Fanuc TP program (LS listing): pick_and_place.ls

/PROG  PICK_AND_PLACE
/ATTR
OWNER		= MNEDITOR;
COMMENT		= "";
PROG_SIZE	= 5834;
CREATE		= DATE 26-07-14  TIME 16:19:38;
MODIFIED	= DATE 26-07-14  TIME 16:19:38;
FILE_NAME	= PICK_AND;
VERSION		= 0;
LINE_COUNT	= 270;
MEMORY_SIZE	= 6422;
PROTECT		= READ_WRITE;
TCD:  STACK_SIZE	= 0,
      TASK_PRIORITY	= 50,
      TIME_SLICE	= 0,
      BUSY_LAMP_OFF	= 0,
      ABORT_REQUEST	= 0,
      PAUSE_REQUEST	= 0;
DEFAULT_GROUP	= 1,*,*,*,*;
CONTROL_CODE	= 00000000 00000000;
LOCAL_REGISTERS	= 0,0,0;
/APPL
/APPL
/MN
   1:  ! Main driving loop ;
   2:  LBL[4:PP_LOOP] ;
   3:   ;
   4:  ! Reset Error Checking ;
   5:  R[24:PICK_CNT_ERR]=0    ;
   6:  R[25:PLACE_CNT_ERR]=0    ;
   7:   ;
   8:  ! Check for recipe reset ;
   9:  IF R[11:RECIPE_IO_IDX]=37,JMP LBL[998] ;
  10:  R[12:RECIPE_OUTPUT]=R[R[99]]    ;
  11:   ;
  12:  ! Checks next recipe output ;
  13:  IF R[12:RECIPE_OUTPUT]=0,JMP LBL[1] ;
  14:   ;
  15:  LBL[24] ;
  16:  ! get out of shroud safely ;
  17:J PR[20] 100% CNT30    ;
  18:   ;
  19:  ! Move to next pin ;
  20:J PR[5:REPO_RCP_PSN] 100% FINE    ;
  21:   ;
  22:  ! Descend to grab pin ;
  23:  PR[2:TMP_REPO_RCP]=PR[5:REPO_RCP_PSN]    ;
  24:  PR[2,3:TMP_REPO_RCP]=PR[2,3:TMP_REPO_RCP]-R[21:PICKUP_CONSTANT]    ;
  25:L PR[2:TMP_REPO_RCP] 100mm/sec FINE    ;
  26:   ;
  27:  ! Ascend with Pin ;
  28:L PR[5:REPO_RCP_PSN] 100mm/sec FINE    ;
  29:   ;
  30:  ! Move safely to shroud ;
  31:  PR[20]=PR[5:REPO_RCP_PSN]    ;
  32:  PR[20,3]=PR[3,3:TMP_CAMERA]    ;
  33:  PR[20,1]=PR[3,1:TMP_CAMERA]    ;
  34:J PR[20] 100% CNT30    ;
  35:J PR[3:TMP_CAMERA] 100% FINE    ;
  36:   ;
  37:   ;
  38:   ;
  39:  ! initiate camera code ;
  40:  R[50:STEP_CNT]=0    ;
  41:  R[51:MAX_STEP_CNT]=47    ;
  42:  R[52:TURN_PER_STEP]=8    ;
  43:  R[53:MINIMUM_THRESH]=90    ;
  44:  R[54:ABOVE_THRESH]=0    ;
  45:  R[55:BEST_SCORE]=0    ;
  46:  R[56:DOWN_THRESH]=2    ;
  47:  R[57:CUR_SCORE]=0    ;
  48:  R[58:CUR_DROP]=0    ;
  49:  PR[21]=PR[3:TMP_CAMERA]    ;
  50:  PR[22]=PR[3:TMP_CAMERA]    ;
  51:   ;
  52:   ;
  53:  CALL READ_SCORE    ;
  54:  IF R[57:CUR_SCORE]>0,JMP LBL[30] ;
  55:  MESSAGE[FAILED PICK] ;
  56:  IF R[25:PLACE_CNT_ERR]=3,JMP LBL[38] ;
  57:  R[24:PICK_CNT_ERR]=R[24:PICK_CNT_ERR]+1    ;
  58:  JMP LBL[24] ;
  59:   ;
  60:  ! FIND BEST ORIENTATION ;
  61:  ! Rotate to next step ;
  62:  LBL[30] ;
  63:  R[24:PICK_CNT_ERR]=0    ;
  64:L PR[21] 1000deg/sec FINE    ;
  65:  WAIT    .02(sec) ;
  66:  CALL READ_SCORE    ;
  67:  IF R[57:CUR_SCORE]>R[55:BEST_SCORE],JMP LBL[31] ;
  68:  IF R[54:ABOVE_THRESH]=1,JMP LBL[33] ;
  69:  JMP LBL[34] ;
  70:   ;
  71:  ! Entered quality threshold ;
  72:  LBL[31] ;
  73:  R[55:BEST_SCORE]=R[57:CUR_SCORE]    ;
  74:  PR[22]=PR[21]    ;
  75:  IF R[57:CUR_SCORE]>R[53:MINIMUM_THRESH],JMP LBL[32] ;
  76:  JMP LBL[34] ;
  77:   ;
  78:  ! In quality threshold - NEW BEST ;
  79:  LBL[32] ;
  80:  R[54:ABOVE_THRESH]=1    ;
  81:  JMP LBL[34] ;
  82:   ;
  83:  ! Significant downturn check ;
  84:  LBL[33] ;
  85:  R[58:CUR_DROP]=R[55:BEST_SCORE]-R[57:CUR_SCORE]    ;
  86:  IF R[58:CUR_DROP]>R[56:DOWN_THRESH],JMP LBL[35] ;
  87:  JMP LBL[34] ;
  88:   ;
  89:  ! Iterate and call next step ;
  90:  LBL[34] ;
  91:  R[50:STEP_CNT]=R[50:STEP_CNT]+1    ;
  92:  IF R[50:STEP_CNT]>=R[51:MAX_STEP_CNT],JMP LBL[37] ;
  93:  PR[21,6]=PR[21,6]+R[52:TURN_PER_STEP]    ;
  94:  JMP LBL[30] ;
  95:   ;
  96:  ! Found Peak or no match ;
  97:  LBL[35] ;
  98:J PR[22] 100% CNT30    ;
  99:  JMP LBL[36] ;
 100:   ;
 101:  ! Fail Case: No Match ;
 102:  LBL[37] ;
 103:  MESSAGE[NO HIGH MATCH] ;
 104:J PR[22] 100% CNT30    ;
 105:  JMP LBL[36] ;
 106:   ;
 107:  ! Done (don't forget to maintain ;
 108:  ! rotation values ;
 109:  LBL[36] ;
 110:  PR[6,6:MOD_RCP_PSN]=PR[22,6]    ;
 111:   ;
 112:  ! Move out of shroud ;
 113:  PR[20]=PR[3:TMP_CAMERA]    ;
 114:  PR[20,2]=PR[20,2]-R[23:Y_OFFSET_SHROUD]    ;
 115:  PR[20,6]=PR[22,6]    ;
 116:  LBL[25] ;
 117:J PR[20] 100% CNT30    ;
 118:   ;
 119:  ! Move to Cable Module ;
 120:J PR[6:MOD_RCP_PSN] 100% FINE    ;
 121:   ;
 122:  ! Descend with receptacle ;
 123:  PR[4:TMP_MOD_RCP]=PR[6:MOD_RCP_PSN]    ;
 124:  PR[4,3:TMP_MOD_RCP]=PR[4,3:TMP_MOD_RCP]-R[22:RELEASE_CONSTANT]    ;
 125:L PR[4:TMP_MOD_RCP] 100mm/sec FINE    ;
 126:   ;
 127:  ! Ascend without receptacle ;
 128:L PR[6:MOD_RCP_PSN] 100mm/sec FINE    ;
 129:  ! Move safely back to shroud ;
 130:J PR[20] 100% CNT30    ;
 131:  ! Check without receptacle ;
 132:  R[57:CUR_SCORE]=0    ;
 133:J PR[22] 100% FINE    ;
 134:  CALL READ_SCORE    ;
 135:  IF R[57:CUR_SCORE]=0,JMP LBL[38] ;
 136:  IF R[25:PLACE_CNT_ERR]=3,JMP LBL[28] ;
 137:  R[25:PLACE_CNT_ERR]=R[25:PLACE_CNT_ERR]+1    ;
 138:  JMP LBL[25] ;
 139:   ;
 140:  LBL[28] ;
 141:  ! Put pin extraction code here. ;
 142:J PR[20] 100% CNT30    ;
 143:J PR[25] 100% CNT30    ;
 144:J PR[26] 100% CNT30    ;
 145:  MESSAGE[PLACE FAILED CLEAR PART RESUME] ;
 146:  PAUSE ;
 147:J PR[25] 100% CNT30    ;
 148:J PR[20] 100% CNT30    ;
 149:   ;
 150:   ;
 151:  !!! CHECK REPO STATUS START ;
 152:  LBL[38] ;
 153:  IF R[1:REPO_RCP_X]=22 AND R[2:REPO_RCP_Y]=20,JMP LBL[999] ;
 154:   ;
 155:  ! Not empty so update ;
 156:  R[1:REPO_RCP_X]=R[1:REPO_RCP_X]+1    ;
 157:  IF R[1:REPO_RCP_X]>22,JMP LBL[2] ;
 158:   ;
 159:  ! Update position x ;
 160:  PR[5,1:REPO_RCP_PSN]=PR[5,1:REPO_RCP_PSN]+R[3:REPO_RCP_UOFFSET]    ;
 161:  JMP LBL[1] ;
 162:   ;
 163:  ! Next row x overflow ;
 164:  LBL[2] ;
 165:  R[1:REPO_RCP_X]=1    ;
 166:  R[2:REPO_RCP_Y]=R[2:REPO_RCP_Y]+1    ;
 167:  PR[5,1:REPO_RCP_PSN]=PR[9,1:REPO_PSN]    ;
 168:  PR[5,2:REPO_RCP_PSN]=PR[5,2:REPO_RCP_PSN]-R[3:REPO_RCP_UOFFSET]    ;
 169:  JMP LBL[1] ;
 170:   ;
 171:  ! Switched from receptacle repo ;
 172:  ! to receptacle repo ;
 173:  LBL[999] ;
 174:  R[1:REPO_RCP_X]=1    ;
 175:  R[2:REPO_RCP_Y]=1    ;
 176:  IF R[4:REPO_X]=2 AND R[18:REPO_Y]=2,JMP LBL[996] ;
 177:   ;
 178:  R[4:REPO_X]=R[4:REPO_X]+1    ;
 179:  IF R[4:REPO_X]>2,JMP LBL[7] ;
 180:   ;
 181:  ! next repository column ;
 182:  PR[9,1:REPO_PSN]=PR[9,1:REPO_PSN]+R[19:REPO_XOFFSET]    ;
 183:  PR[5:REPO_RCP_PSN]=PR[9:REPO_PSN]    ;
 184:  JMP LBL[1] ;
 185:   ;
 186:  ! next repository row ;
 187:  LBL[7] ;
 188:  R[4:REPO_X]=1    ;
 189:  R[18:REPO_Y]=R[18:REPO_Y]+1    ;
 190:  PR[9,1:REPO_PSN]=PR[7,1:TMP_REPO_RCP]    ;
 191:  PR[9,2:REPO_PSN]=PR[9,2:REPO_PSN]-R[20:REPO_YOFFSET]    ;
 192:  PR[5:REPO_RCP_PSN]=PR[9:REPO_PSN]    ;
 193:  JMP LBL[1] ;
 194:  !!! CHECK REPO STATUS END. ;
 195:   ;
 196:   ;
 197:   ;
 198:  !!! CHECK TO SEE CURRENT RECIPE S ;
 199:  LBL[1] ;
 200:  IF R[24:PICK_CNT_ERR]=3,JMP LBL[4] ;
 201:  IF R[25:PLACE_CNT_ERR]=3,JMP LBL[4] ;
 202:  R[11:RECIPE_IO_IDX]=R[11:RECIPE_IO_IDX]+1    ;
 203:  R[99:RECIPE_IDX]=R[99:RECIPE_IDX]+1    ;
 204:  R[8:MOD_RCP_X]=R[8:MOD_RCP_X]+1    ;
 205:   ;
 206:  IF R[8:MOD_RCP_X]>6,JMP LBL[5] ;
 207:   ;
 208:  PR[6,1:MOD_RCP_PSN]=PR[6,1:MOD_RCP_PSN]+R[6:MOD_RCP_XOFFSET]    ;
 209:  JMP LBL[4] ;
 210:   ;
 211:  LBL[5] ;
 212:  R[8:MOD_RCP_X]=1    ;
 213:  R[9:MOD_RCP_Y]=R[9:MOD_RCP_Y]+1    ;
 214:  PR[6,1:MOD_RCP_PSN]=PR[8,1:MOD_PSN]    ;
 215:  PR[6,2:MOD_RCP_PSN]=PR[6,2:MOD_RCP_PSN]-R[7:MOD_RCP_YOFFSET]    ;
 216:  JMP LBL[4] ;
 217:  !!! CHECK TO SEE CURRENT RECIPE ;
 218:  !!! END ;
 219:   ;
 220:   ;
 221:   ;
 222:  !!! MODULE FULL, CHECK STATUS ;
 223:  !!! START ;
 224:  LBL[998] ;
 225:  R[11:RECIPE_IO_IDX]=1    ;
 226:  R[99:RECIPE_IDX]=101    ;
 227:  R[8:MOD_RCP_X]=1    ;
 228:  R[9:MOD_RCP_Y]=1    ;
 229:   ;
 230:  ! Check to see if Ice Tray Full ;
 231:  IF R[5:MODULE_X]=6 AND R[15:MODULE_Y]=4,JMP LBL[997] ;
 232:   ;
 233:  ! Check if module row full ;
 234:  R[5:MODULE_X]=R[5:MODULE_X]+1    ;
 235:  IF R[5:MODULE_X]>6,JMP LBL[6] ;
 236:   ;
 237:  ! Increment module column ;
 238:  PR[8,1:MOD_PSN]=PR[8,1:MOD_PSN]+R[13:MODULE_XOFFSET]    ;
 239:  PR[6:MOD_RCP_PSN]=PR[8:MOD_PSN]    ;
 240:  JMP LBL[4] ;
 241:   ;
 242:  ! Increment module row and reset  ;
 243:  LBL[6] ;
 244:  R[5:MODULE_X]=1    ;
 245:  R[15:MODULE_Y]=R[15:MODULE_Y]+1    ;
 246:  PR[8,1:MOD_PSN]=PR[10,1:TMP_MOD_RCP]    ;
 247:  PR[8,2:MOD_PSN]=PR[8,2:MOD_PSN]-R[14:MODULE_YOFFSET]    ;
 248:  PR[6:MOD_RCP_PSN]=PR[8:MOD_PSN]    ;
 249:  JMP LBL[4] ;
 250:   ;
 251:  ! Switched from ice tray ;
 252:  ! to ice tray ;
 253:  LBL[997] ;
 254:  ! Check am I out of Ice Trays ;
 255:  IF R[16:ICE_TRAY_NUM]=2,JMP LBL[996] ;
 256:   ;
 257:  ! Increment Ice Tray and set mod ;
 258:  ! and mod_rcp equal ;
 259:  R[5:MODULE_X]=1    ;
 260:  R[15:MODULE_Y]=1    ;
 261:  R[16:ICE_TRAY_NUM]=R[16:ICE_TRAY_NUM]+1    ;
 262:  PR[11,2:ICE_TRAY_PSN]=PR[11,2:ICE_TRAY_PSN]-R[17:ICE_TRAY_YOFFSET]    ;
 263:  PR[8:MOD_PSN]=PR[11:ICE_TRAY_PSN]    ;
 264:  PR[6:MOD_RCP_PSN]=PR[8:MOD_PSN]    ;
 265:  JMP LBL[4] ;
 266:  !!! MODULE FULL, CHECK STATUS ;
 267:  !!! END ;
 268:   ;
 269:  LBL[996] ;
 270:  END ;
/POS
P[1:"DATUM"]{
   GP1:
	UF : 1, UT : 1,		CONFIG : 'L, 0, 0, 0',
	X =   424.654999  mm,	Y =   183.154999  mm,	Z =     0.000000  mm,
	W =  -180.000000 deg,	P =     0.000000 deg,	R =     0.000000 deg
};
P[2:"FIRST_PIN"]{
   GP1:
	UF : 1, UT : 1,		CONFIG : 'L, 0, 0, 0',
	X =   369.580994  mm,	Y =   174.535004  mm,	Z =     0.000000  mm,
	W =  -180.000000 deg,	P =     0.000000 deg,	R =     0.000000 deg
};
P[3:"CAMERA"]{
   GP1:
	UF : 1, UT : 1,		CONFIG : 'L, 0, 0, 0',
	X =   207.901993  mm,	Y =   332.035004  mm,	Z =    82.065002  mm,
	W =  -180.000000 deg,	P =     0.000000 deg,	R =     0.000000 deg
};
P[4:"FIRST_RCP"]{
   GP1:
	UF : 1, UT : 1,		CONFIG : 'L, 0, 0, 0',
	X =   108.552002  mm,	Y =   190.020996  mm,	Z =     0.000000  mm,
	W =  -180.000000 deg,	P =     0.000000 deg,	R =     0.000000 deg
};
/END
